// TIA Portal V18 export
FUNCTION_BLOCK "AndonBoxASi"   // FB13, FBD
{ S7_Optimized_Access := 'TRUE' }
VERSION : 0.1
// stored: AutoNumber true, IsIECCheckEnabled false, IsRetainMemResEnabled false, MemoryReserve 100, SetENOAutomatically false, UDAEnableTagReadback false
   VAR_INPUT
      I_greenBtn { ExternalAccessible := 'False'; ExternalVisible := 'False'; ExternalWritable := 'False'} : Bool;
      I_yellowBtn { ExternalAccessible := 'False'; ExternalVisible := 'False'; ExternalWritable := 'False'} : Bool;
      I_redBtn { ExternalAccessible := 'False'; ExternalVisible := 'False'; ExternalWritable := 'False'} : Bool;
      I_FlashingPeriod { ExternalAccessible := 'False'; ExternalVisible := 'False'; ExternalWritable := 'False'} : Time;
      I_greenFlashingDuration { ExternalAccessible := 'False'; ExternalVisible := 'False'; ExternalWritable := 'False'} : Time;
      I_yellowFlashingDuration { ExternalAccessible := 'False'; ExternalVisible := 'False'; ExternalWritable := 'False'} : Time;
      I_redFlashingDuration { ExternalAccessible := 'False'; ExternalVisible := 'False'; ExternalWritable := 'False'} : Time;
   END_VAR
   VAR_OUTPUT
      O_state { ExternalAccessible := 'False'; ExternalVisible := 'False'; ExternalWritable := 'False'} : Int;
      O_greenBtnLed { ExternalAccessible := 'False'; ExternalVisible := 'False'; ExternalWritable := 'False'} : Bool;
      O_yellowBtnLed { ExternalAccessible := 'False'; ExternalVisible := 'False'; ExternalWritable := 'False'} : Bool;
      O_redBtnLed { ExternalAccessible := 'False'; ExternalVisible := 'False'; ExternalWritable := 'False'} : Bool;
   END_VAR
   VAR_IN_OUT
      IO_sireneGreenTrigger { ExternalAccessible := 'False'; ExternalVisible := 'False'; ExternalWritable := 'False'} : Bool;
      IO_sireneYellowTrigger { ExternalAccessible := 'False'; ExternalVisible := 'False'; ExternalWritable := 'False'} : Bool;
      IO_sireneRedTrigger { ExternalAccessible := 'False'; ExternalVisible := 'False'; ExternalWritable := 'False'} : Bool;
   END_VAR
   VAR
      fpBit_greenBtn { ExternalAccessible := 'False'; ExternalVisible := 'False'; ExternalWritable := 'False'} : Bool;
      fpBit_yellowBtn { ExternalAccessible := 'False'; ExternalVisible := 'False'; ExternalWritable := 'False'} : Bool;
      fpBit_redBtn { ExternalAccessible := 'False'; ExternalVisible := 'False'; ExternalWritable := 'False'} : Bool;
   END_VAR
   VAR RETAIN
      memState { ExternalAccessible := 'False'; ExternalVisible := 'False'; ExternalWritable := 'False'} : Int;
   END_VAR
   VAR
      IEC_Timer_0_Instance { ExternalAccessible := 'False'; ExternalVisible := 'False'; ExternalWritable := 'False'; S7_SetPoint := 'True'} : TP_TIME;
      BtnLedAppearance_Instance { ExternalAccessible := 'False'; ExternalVisible := 'False'; ExternalWritable := 'False'; S7_SetPoint := 'True'} : "BtnLedAppearance";
      BtnLedAppearance_Instance_1 { ExternalAccessible := 'False'; ExternalVisible := 'False'; ExternalWritable := 'False'; S7_SetPoint := 'True'} : "BtnLedAppearance";
      BtnLedAppearance_Instance_2 { ExternalAccessible := 'False'; ExternalVisible := 'False'; ExternalWritable := 'False'; S7_SetPoint := 'True'} : "BtnLedAppearance";
   END_VAR
   VAR_TEMP
      T_fpGreen : Bool;
      T_fpYellow : Bool;
      T_fpRed : Bool;
   END_VAR
   VAR_TEMP   // added for the SCL form of the ladder/FBD networks
      _w1 : Bool;
   END_VAR
BEGIN

REGION Network 1: positive edge green button
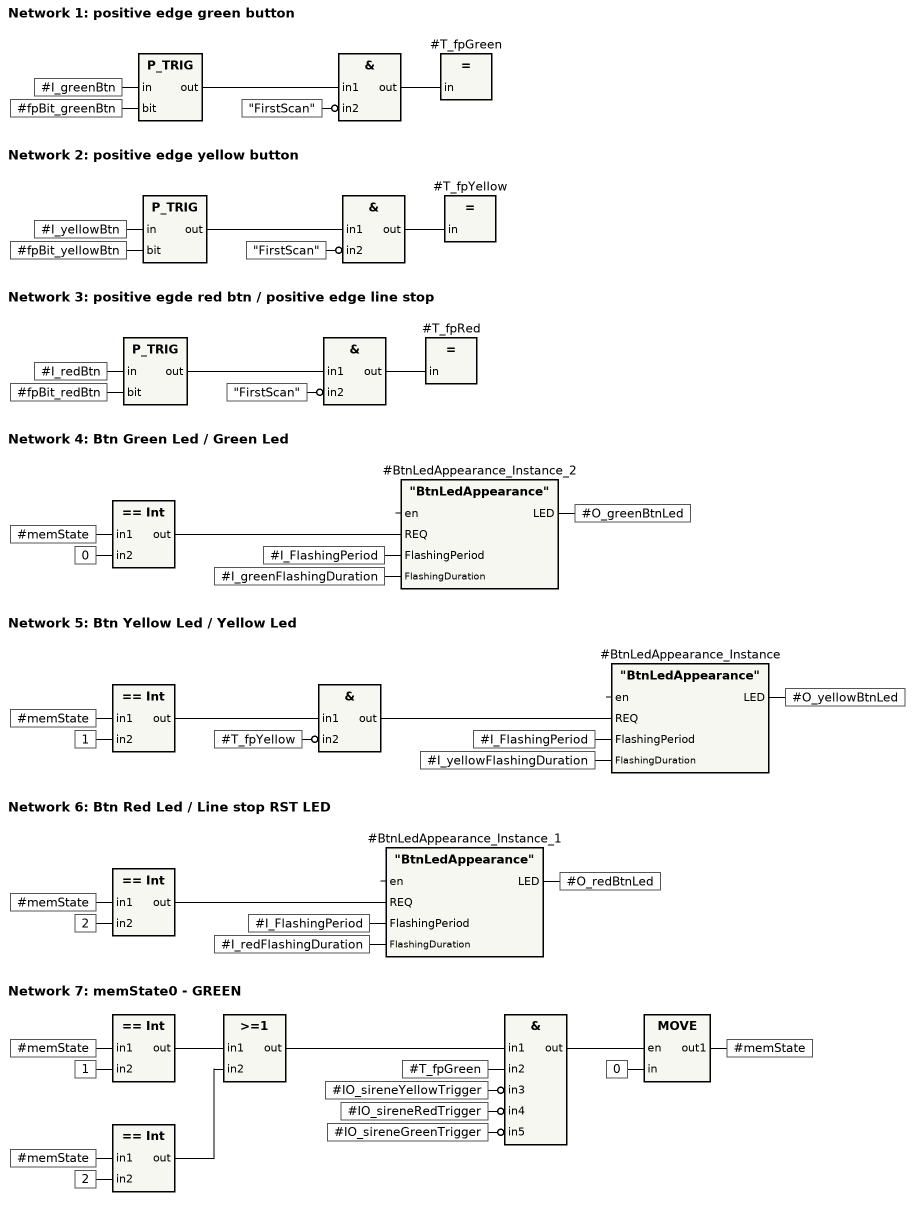
   #_w1 := #I_greenBtn AND NOT #fpBit_greenBtn;   // rising edge
   #fpBit_greenBtn := #I_greenBtn;
   #T_fpGreen := #_w1 AND NOT "FirstScan";
END_REGION

REGION Network 2: positive edge yellow button
   #_w1 := #I_yellowBtn AND NOT #fpBit_yellowBtn;   // rising edge
   #fpBit_yellowBtn := #I_yellowBtn;
   #T_fpYellow := #_w1 AND NOT "FirstScan";
END_REGION

REGION Network 3: positive egde red btn / positive edge line stop
   #_w1 := #I_redBtn AND NOT #fpBit_redBtn;   // rising edge
   #fpBit_redBtn := #I_redBtn;
   #T_fpRed := #_w1 AND NOT "FirstScan";
END_REGION

REGION Network 4: Btn Green Led / Green Led
   #BtnLedAppearance_Instance_2(REQ := #memState = 0,   // "BtnLedAppearance"
                           FlashingPeriod := #I_FlashingPeriod,
                           FlashingDuration := #I_greenFlashingDuration,
                           LED => #O_greenBtnLed);
END_REGION

REGION Network 5: Btn Yellow Led / Yellow Led
   #BtnLedAppearance_Instance(REQ := (#memState = 1) AND NOT #T_fpYellow,   // "BtnLedAppearance"
                           FlashingPeriod := #I_FlashingPeriod,
                           FlashingDuration := #I_yellowFlashingDuration,
                           LED => #O_yellowBtnLed);
END_REGION

REGION Network 6: Btn Red Led / Line stop RST LED
   #BtnLedAppearance_Instance_1(REQ := #memState = 2,   // "BtnLedAppearance"
                           FlashingPeriod := #I_FlashingPeriod,
                           FlashingDuration := #I_redFlashingDuration,
                           LED => #O_redBtnLed);
END_REGION

REGION Network 7: memState0 - GREEN
   IF ((#memState = 1) OR (#memState = 2)) AND #T_fpGreen AND NOT #IO_sireneYellowTrigger AND NOT #IO_sireneRedTrigger AND NOT #IO_sireneGreenTrigger THEN
       #memState := 0;
   END_IF;
END_REGION

REGION Network 8: memState1 - YELLOW / Yellow button / State1
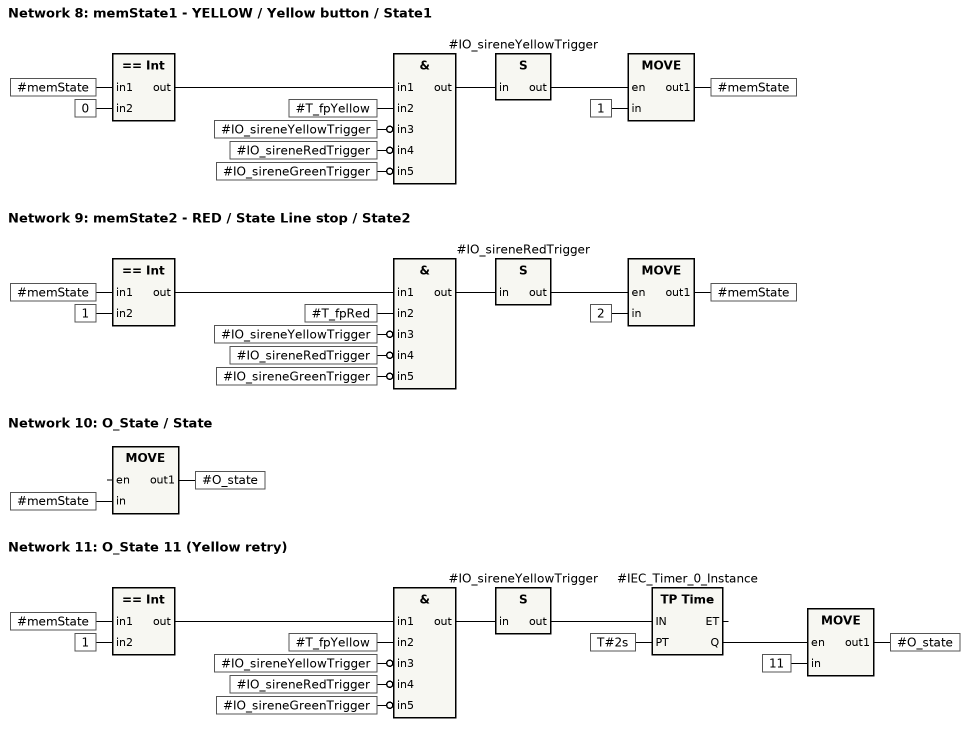
   #_w1 := (#memState = 0) AND #T_fpYellow AND NOT #IO_sireneYellowTrigger AND NOT #IO_sireneRedTrigger AND NOT #IO_sireneGreenTrigger;
   IF #_w1 THEN
       #IO_sireneYellowTrigger := TRUE;
       #memState := 1;
   END_IF;
END_REGION

REGION Network 9: memState2 - RED / State Line stop / State2
   #_w1 := (#memState = 1) AND #T_fpRed AND NOT #IO_sireneYellowTrigger AND NOT #IO_sireneRedTrigger AND NOT #IO_sireneGreenTrigger;
   IF #_w1 THEN
       #IO_sireneRedTrigger := TRUE;
       #memState := 2;
   END_IF;
END_REGION

REGION Network 10: O_State / State
   #O_state := #memState;
END_REGION

REGION Network 11: O_State 11 (Yellow retry)
   #_w1 := (#memState = 1) AND #T_fpYellow AND NOT #IO_sireneYellowTrigger AND NOT #IO_sireneRedTrigger AND NOT #IO_sireneGreenTrigger;
   IF #_w1 THEN #IO_sireneYellowTrigger := TRUE; END_IF;
   #IEC_Timer_0_Instance(IN := #_w1, PT := T#2s);   // TP
   IF #IEC_Timer_0_Instance.Q THEN #O_state := 11; END_IF;
END_REGION
END_FUNCTION_BLOCK
